		6:
			// Entry action
			IF (stStatemachine.uinState_old <> stStatemachine.uinState) THEN
				//*********************************************************
				// file close
				fbFileClose.sNetId := ''; // only local access
				fbFileClose.hFile := fbFileOpen.hFile; // only local access
				fbFileClose.tTimeout := T#3S;
				fbFileClose(bExecute:= FALSE);
				fbFileClose(bExecute:= TRUE);
				udiWaitFileCloseCycles := 0;
					
				 stStatemachine.uinState_old := stStatemachine.uinState;
			END_IF
				
			// wait UNTIL closed
			IF (fbFileClose.bBusy) THEN
				udiWaitFileCloseCycles := udiWaitFileCloseCycles + 1;
				fbFileClose(bExecute:=FALSE);
			ELSE
				IF fbFileClose.bError THEN
					strInfo := 'template/config file close failed';
					Out_udiStatus := fbFileClose.nErrId;
					RETURN;
				END_IF
				
				// delocate memory
				__DELETE(pDelReadPointer);
				
				// allocat for temporary item list
				// nbr of items * size for value output + nbf of items * Pre- and Post - Text
				// with this calculation is the buffer normally greater than necessary
				// cMAX_ITEM_CHAR has to be defined for worst case (big 4-byt values, date strings) so big
				udiTmpLen := (In_pstSysInfo^.stItemInfo.uinActNbrOfItems*FileLc.cMAX_ITEM_CHAR) + (In_pstSysInfo^.stItemInfo.uinActNbrOfItems*FileLc.cPRE_POST_TEXTLEN);
				In_pstSysInfo^.p_bytTmpRecordText := M_AllocMEM(In_SizeOfBuffer:=UDINT_TO_UINT(udiTmpLen));
				IF (In_pstSysInfo^.p_bytTmpRecordText=TC3_MEMMAN.NULL) THEN
					strInfo := 'template/config file: alloc memory for temp record text failed';
					Out_udiStatus := FileLc.cERR_ALLOC_MEMORY;
					RETURN;
				END_IF
				In_pstSysInfo^.udiTmpRecordSize := udiTmpLen;
				
				// allocat for temporary file buffer
				udiTmpLen := udiTmpLen*FileLc.cMAX_RECORDS_IN_FILE_BUF;
				In_pstSysInfo^.stFileHandler.p_bytTmpFileBuffer := M_AllocMEM(In_SizeOfBuffer:=UDINT_TO_UINT(udiTmpLen));
				IF (In_pstSysInfo^.stFileHandler.p_bytTmpFileBuffer=TC3_MEMMAN.NULL) THEN
					strInfo := 'template/config file: alloc memory for temp file buffer failed';
					Out_udiStatus := FileLc.cERR_ALLOC_MEMORY;
					RETURN;
				END_IF
				In_pstSysInfo^.stFileHandler.udiTmpFileBufferSize := udiTmpLen;
				stStatemachine.uinState := stStatemachine.uinState  + 1;
			END_IF
			
		
		7:
			stStatemachine.usiInitDone := 1;
			Out_bolDone := TRUE;
			strInfo := 'template/config file: successfully parsed';
			Out_udiStatus := 0;
	END_CASE
END_IF
bolExecute_old := In_bolExecute;

METHOD FB_exit : BOOL
VAR_INPUT
	bInCopyCode : BOOL; // if TRUE, the exit method is called for exiting an instance that is copied afterwards (online change).
END_VAR
__DELETE(pDelReadPointer);
END_METHOD

METHOD PROTECTED M_AllocMEM : POINTER TO BYTE

VAR_INPUT
	In_SizeOfBuffer : UINT; // Byte size of quee to allocate
END_VAR
// Debug counter
M_AllocMEM := __NEW(BYTE,In_SizeOfBuffer);

// check if allocate memory is ok
IF (M_AllocMEM=TC3_MEMMAN.NULL) THEN
	M_AllocMEM := TC3_MEMMAN.NULL;
ELSE
	Tc2_System.MEMSET(M_AllocMEM,0,In_SizeOfBuffer); // init with zero.
END_IF
END_METHOD

METHOD M_ReleaseAllMEM : BOOL
VAR_INPUT
	In_pstSysInfo : POINTER TO T_FileLc_SysInfo;
END_VAR
VAR
	pDelPointer : POINTER TO BYTE;
END_VAR
// no usage at the moment -> with handle shutdown sequence no easy to remove every thing in the right order


// the other allocated memory has to be deallocated by FB_FileLC! on exit this methode should be called from FB_FileLC!
IF (In_pstSysInfo<>TC3_MEMMAN.NULL) THEN
	__DELETE(In_pstSysInfo^.p_bytHeaderText);
	__DELETE(In_pstSysInfo^.p_bytFooterText);
	FOR ii:=0 TO Queue.cMAX_NR_OF_TASKS BY 1 DO
		IF (In_pstSysInfo^.stItemInfo.a_p_bytItemDataList[ii]<>TC3_MEMMAN.NULL) THEN
			pDelPointer := In_pstSysInfo^.stItemInfo.a_p_bytItemDataList[ii];
			__DELETE(pDelPointer);
			In_pstSysInfo^.stItemInfo.a_p_bytItemDataList[ii] := 0;
		END_IF
	END_FOR
	__DELETE(In_pstSysInfo^.stItemInfo.p_bytItemCfgList);
	__DELETE(In_pstSysInfo^.p_bytTmpRecordText);
	__DELETE(In_pstSysInfo^.stFileHandler.p_bytTmpFileBuffer);
	__DELETE(pDelReadPointer);
END_IF
END_METHOD

END_FUNCTION_BLOCK

// POUs/Utility/strstr
FUNCTION strstr : POINTER TO BYTE
VAR_INPUT
	In_pStr: POINTER TO BYTE; // string which should include search string
	In_pStrSearch: POINTER TO BYTE; // search string
	In_bolAddStrSearchLen : BOOL; // add to result search STRING length
END_VAR
VAR
	p_bytStr : POINTER TO BYTE;
	chrStr : STRING(1) := '';
	p_bytStrSearch : POINTER TO BYTE;
	chrStrSearch : STRING(1) := '';
	ii : UINT;
	jj : UINT;
	p_bytAdressStr : POINTER TO BYTE;
	p_bytAdressStrSearch : POINTER TO BYTE;
END_VAR

(*char *strstr(const char *s1, const char *s2);

Description
Locates the first occurence in the string pointed to by s1 of the sequence of characters in the string pointed to by s2 (excluding the terminating null character). 


Returns
Returns a pointer to the located string segment, or a null pointer if the string s2 is not found. If s2 points to a string with zero length, the s1 is returned. 
*)

// invalid input pointer check
IF ((In_pStr=TC3_MEMMAN.NULL) OR (In_pStrSearch=TC3_MEMMAN.NULL)) THEN
	strstr := TC3_MEMMAN.NULL; // input strings not defined
	RETURN;
END_IF


ii :=0;
p_bytAdressStr := In_pStr;
p_bytStr := p_bytAdressStr;
WHILE (p_bytStr^ <> 0) DO // zero terminated string
	p_bytAdressStr := In_pStr + ii*SIZEOF(In_pStr^); // pointer increment
	p_bytStr := p_bytAdressStr;
	chrStr :=Tc2_System.F_ToCHR(c:= p_bytStr^); // for debugging watch value
	
	jj := 0;
	p_bytAdressStrSearch := In_pStrSearch;
	p_bytStrSearch := p_bytAdressStrSearch;

	WHILE (p_bytStr^ = p_bytStrSearch^) DO
		
		// char/byte matches compare next
		p_bytAdressStrSearch := In_pStrSearch + jj*SIZEOF(In_pStrSearch^); // pointer increment
		p_bytStrSearch := p_bytAdressStrSearch;
		chrStrSearch := Tc2_System.F_ToCHR(c:= p_bytStrSearch^); // for debugging watch value
		
		// end of string found->search string matches
		IF (p_bytStrSearch^=0) THEN// zero terminated string
			IF (In_bolAddStrSearchLen=TRUE) THEN// add to result search STRING length
				strstr := p_bytAdressStr + jj*SIZEOF(In_pStr^); // return start adress of next byte after search string
			ELSE
				strstr := p_bytAdressStr; // return start adress of match search string
			END_IF
			
			RETURN;
		END_IF
		
		p_bytStr := p_bytAdressStr + jj*SIZEOF(In_pStr^);
		chrStr :=Tc2_System.F_ToCHR(c:= p_bytStr^); // for debugging watch value
		jj := jj + 1;
	END_WHILE
	ii := ii + 1;
END_WHILE

strstr := Tc3_MemMan.NULL; // return null adress search string not found in string

END_FUNCTION

// POUs/Utility/Logger/FileLc/FB_FileLcTest
FUNCTION_BLOCK FB_FileLcTest
VAR_INPUT
	In_p_fbBasLog: POINTER TO FB_BasLog; // only one central FB_BasLog instance allowed per PLC!!!
	In_p_fbFileLC: POINTER TO FB_FileLc; // only one central FB_FileLc instance allowed per PLC!!!
	In_strPath: STRING(FileLc.cPATH_LENGTH); //'C:\Vistaprint\Log\'
	In_strCfgFileName: STRING(FileLc.cFILENAME_LENGTH); // 'StateLogTest.cfg'
END_VAR
VAR_OUTPUT
	Out_bolInitDone : BOOL;
	Out_udiStatus : UDINT;
END_VAR
VAR
	bolGetFirstHandle : BOOL;
	bolDone : BOOL;
	udiInitStatus : UDINT;
	udiStatus : UDINT;
	pHandle : POINTER TO T_FileLc_SysInfo;
	// for test send
	pHandleBaseLog : POINTER TO T_Bl_LibHandleRow;
	uinGetHandleBaseLogStatus : UINT;
	intDoWrite : INT;
	dinPar1 : DINT;
	strText1 : STRING(30):='Controller 1';
	strText2 : STRING(30):='Alarm sub info';
	uinWriteStatus : UINT;
	bolStressTest : BOOL;
	fbRAND : DRAND;
	uinActFLcClientIdx : UINT; // file client index for init
END_VAR

(*__________________________________________________________________________________________________
¦	
¦	Vistaprint Schweiz GmbH
¦	CH - 8401 Winterthur
¦
¦	www.vistaprint.ch - info@vistaprint.ch
¦___________________________________________________________________________________________________

Function desription:
Function block capsule the logger file client call for tests.

History:
Version		Date			Author		Comment
---------------------------------------------------------------------------------------------------
0.00.1		27.10.2014		AVME/KVO	Start history
___________________________________________________________________________________________________*)

IF (In_p_fbFileLC<>TC3_MEMMAN.NULL) THEN // check if pointer valid
	
	// system init onetime after start up
	IF (Out_bolInitDone=FALSE) THEN
		In_p_fbFileLC^.M_Init(In_bolExecute := TRUE,In_p_uinFLcIdx := ADR(uinActFLcClientIdx),In_strCfgFileName:=In_strCfgFileName ,In_strPath:= In_strPath,In_p_fbBasLog := In_p_fbBasLog,Out_pHandle=>pHandle,Out_udiStatus=>udiInitStatus,Out_bolDone=>bolDone);
		IF (bolDone OR (udiInitStatus<>0)) THEN
			// negative edge -> reinit possibel and release init next file client!!!
			In_p_fbFileLC^.M_Init(In_bolExecute := FALSE,In_p_uinFLcIdx := ADR(uinActFLcClientIdx),In_strCfgFileName:=In_strCfgFileName,In_strPath:=In_strPath,In_p_fbBasLog := In_p_fbBasLog);
			Out_bolInitDone := TRUE;
		END_IF
	ELSE
		IF ((pHandle<>TC3_MEMMAN.NULL) AND (udiInitStatus=0)) THEN	// valid pointer => init ok
			// cyclic call of file client - alarm generation in application if status not ok???
			udiStatus := In_p_fbFileLC^.M_Cyclic(In_pHandle:=pHandle);
			
			// *******************************************************************************************************************************************
			// only for sending test logs!!!
			// get write handle for tests
			IF (bolGetFirstHandle=FALSE) THEN
				uinGetHandleBaseLogStatus := In_p_fbBasLog^.M_GetHandle(Out_pHandle=>pHandleBaseLog);// fbBasLog global defined base log system fub (only once per system)
				bolGetFirstHandle := TRUE;
			END_IF
			
			// write test state log entries
			IF (pHandleBaseLog<>TC3_MEMMAN.NULL) AND (intDoWrite>0) THEN
				intDoWrite := intDoWrite - 1;
				dinPar1 := dinPar1 + 1;
				uinWriteStatus := In_p_fbBasLog^.M_Log(In_pHandle:=pHandleBaseLog,In_udiLogType:=BasLog.cLOGTYPE_STATELOG,In_intCtrlID:=11,In_strText1:=strText1,In_strText2:=strText2,In_dinPar1:=dinPar1,In_dinPar2:=0,In_dinPar3:=0,In_dinPar4:=0) ;
			END_IF
			IF (bolStressTest) THEN
				IF (intDoWrite = 0) THEN
					fbRAND();
					intDoWrite := LREAL_TO_INT(fbRAND.Num*100.0);
					uinWriteStatus := In_p_fbBasLog^.M_Log(In_pHandle:=pHandleBaseLog,In_udiLogType:=BasLog.cLOGTYPE_STATELOG,In_intCtrlID:=intDoWrite,In_strText1:=strText1,In_strText2:=strText2,In_dinPar1:=dinPar1,In_dinPar2:=0,In_dinPar3:=0,In_dinPar4:=0) ;
				END_IF
			END_IF
			// *******************************************************************************************************************************************
		END_IF;		
	END_IF

	// out for failures
	IF (udiInitStatus<>0)THEN
		Out_udiStatus := udiInitStatus;
	ELSE
		Out_udiStatus := udiStatus;
	END_IF
END_IF

END_FUNCTION_BLOCK

// POUs/Utility/Queue/FB_QueueTest_Receiver
FUNCTION_BLOCK FB_QueueTest_Receiver
VAR_INPUT
	In_p_fbQueue: POINTER TO FB_Queue; // only one central FB_QUEUE instance allowed per PLC!!!
END_VAR
VAR_OUTPUT
END_VAR
VAR
	stData : T_Queue_TestData;
	bolInit : BOOL := FALSE;
	pQueueHandle : POINTER TO T_Queue_SysInfo;
	pQueueHandleRead : POINTER TO T_Queue_Info;
	uinInitStatus : UINT;
	uinGetHandleStatus :UINT;
	uinReadStatus : UINT;
	ii:UINT;
	udiRxCounter : UDINT;
END_VAR

(*__________________________________________________________________________________________________
¦	
¦	Vistaprint Schweiz GmbH
¦	CH - 8401 Winterthur
¦
¦	www.vistaprint.ch - info@vistaprint.ch
¦___________________________________________________________________________________________________

Function desription:
Example and test programm for testing the queue system - read data from queue

History:
Version		Date			Author		Comment
---------------------------------------------------------------------------------------------------
0.00.1		14.07.2014		AVME/KVO	Start history
___________________________________________________________________________________________________*)

// system init onetime after start up
IF (bolInit=FALSE) THEN
	//init queue system, one time should be called per queue system
	In_p_fbQueue^.M_Init(In_strQueueName:='bReceiver',In_uinNrOfElement := 25, In_udiSizeOfElement:= SIZEOF(stData),In_uinMode:=0,Out_pHandle=>pQueueHandle,Out_uinStatus=>uinInitStatus);
	
	// for every task class has to call this methode handle is needed for read
	uinGetHandleStatus := In_p_fbQueue^.M_GetHandle(In_strQueueName:='bReceiver',Out_pQueueHandle=>pQueueHandleRead);
	bolInit := TRUE;
END_IF

// because more than one task function writes to the logsystem it is better to read out more than one elment per cycle!
FOR ii:=0 TO 9 BY 1 DO
	uinReadStatus := In_p_fbQueue^.M_Read(In_pQueueHandle:=pQueueHandleRead,In_pData:=ADR(stData));
	IF (uinReadStatus<>0) THEN
		EXIT;
	END_IF
	udiRxCounter := udiRxCounter + 1;
END_FOR

END_FUNCTION_BLOCK

// POUs/Utility/Queue/FB_QueueTest_Sender
FUNCTION_BLOCK FB_QueueTest_Sender
VAR_INPUT
	In_p_fbQueue: POINTER TO FB_Queue; // only one central FB_QUEUE instance allowed per PLC!!!
END_VAR
VAR_OUTPUT
END_VAR
VAR
	stData : T_Queue_TestData;
	bolInit : BOOL := FALSE;
	pQueueHandle : POINTER TO T_Queue_Info;
	uinGetHandleStatus : UINT;
	uinWriteStatus :UINT;
	uinDoWrite : UINT;
END_VAR

(*__________________________________________________________________________________________________
¦	
¦	Vistaprint Schweiz GmbH
¦	CH - 8401 Winterthur
¦
¦	www.vistaprint.ch - info@vistaprint.ch
¦___________________________________________________________________________________________________

Function desription:
Example and test programm for testing the queue system - write data in queue

History:
Version		Date			Author		Comment
---------------------------------------------------------------------------------------------------
0.00.1		14.07.2014		AVME/KVO	Start history
___________________________________________________________________________________________________*)

// system init onetime after start up
IF (bolInit=FALSE) THEN
	uinGetHandleStatus := In_p_fbQueue^.M_GetHandle(In_strQueueName:='bReceiver',Out_pQueueHandle=>pQueueHandle);
	
	// init write struct
	stData.strName := 'Daten';
	stData.udiAdress := 1;
	stData.udiDataLen := 2;
	stData.usiDataTyp:= 3;
	stData.udiDimension := 4;
	bolInit := TRUE;
END_IF

// number of cycles to write
IF (uinDoWrite>0) THEN
	uinDoWrite := uinDoWrite - 1;
	uinWriteStatus := In_p_fbQueue^.M_Write(In_pQueueHandle:= pQueueHandle,In_pData:= ADR(stData));
	stData.udiAdress := stData.udiAdress + 1;
END_IF

END_FUNCTION_BLOCK

// POUs/Utility/SaberLogger/helper/cycle_Logger
FUNCTION cycle_Logger : BOOL
VAR_INPUT
	pLogger			: POINTER TO T_LoggerSendData;
END_VAR
VAR
END_VAR

pLogger^.fbFifo();

END_FUNCTION

// POUs/Utility/SaberLogger/helper/init_Logger
FUNCTION init_Logger : BOOL
VAR_INPUT
	pLogger			: POINTER TO T_LoggerSendData;
END_VAR
VAR
END_VAR

pLogger^.fbDataChannel.InitChannel(SIZEOF(pLogger^.rDataChannelItem), ADR(pLogger^.rDataChannelItem));
pLogger^.fbFifo.DataChannel := ADR(pLogger^.fbDataChannel);
pLogger^.fbFifo.FreeDataPointer := TRUE;
pLogger^.fbFifo.Enable := TRUE;

END_FUNCTION

// POUs/Utility/SaberLogger/FB_LoggerSendDch
FUNCTION_BLOCK FB_LoggerSendDch EXTENDS FB_DataChannelSendBase IMPLEMENTS I_DataChannelSend
VAR
	/// Saber Inteface Variables
	/// -----------------------------------------------------------------
	m_pOutputData: POINTER TO T_Logger_DCH;
END_VAR

SUPER^();

{attribute 'object_name' := 'InitChannel'}
METHOD InitChannel : BOOL
VAR_INPUT
	udiDataSize: UDINT;
	pOutputData: POINTER TO BYTE;
END_VAR
InitChannel := FALSE;

IF udiDataSize > 0 THEN
	IF pOutputData <> TC3_MEMMAN.NULL THEN
		m_uinDataSize := udiDataSize;
		m_pOutputData := pOutputData;
		m_eState := E_PlcSaberDHCState.Init;
		InitChannel := TRUE;
	END_IF
END_IF
END_METHOD

{attribute 'object_name' := 'SendData'}
METHOD SendData : BOOL
VAR_INPUT
	udiDataSize: UDINT;
	pData: POINTER TO BYTE;
END_VAR
SendData := FALSE;

IF m_eState = E_PlcSaberDHCState.WaitForJob THEN
	IF (udiDataSize > 0 ) AND (pData <> TC3_MEMMAN.NULL) THEN
		TC2_SYSTEM.MEMCPY(destAddr := m_pOutputData, srcAddr := pData, n := udiDataSize);
		m_eState := E_PlcSaberDHCState.SendData;	
		SendData := TRUE;
	END_IF	
END_IF
END_METHOD

END_FUNCTION_BLOCK

// POUs/Utility/callAllCtrlInit
FUNCTION callAllCtrlInit : BOOL
VAR_INPUT
	pCtrlInst			: POINTER TO POINTER TO FB_CtrlBase;
	uinCtrlInstLength	: UINT;
END_VAR
VAR
	uinIdx	: UINT;
END_VAR

FOR uinIdx := 0 TO uinCtrlInstLength DO
	IF pCtrlInst[uinIdx] <> 0 THEN
		pCtrlInst[uinIdx]^.CtrlInit(); // init ctrl and add childs
	END_IF
END_FOR

END_FUNCTION

// POUs/Utility/getInBol
FUNCTION getInBol : BOOL
VAR_INPUT
	bol_GlobalEnableForce: BOOL;
	p_Input: POINTER TO T_Ctrl_IoBool;
END_VAR

p_Input^.state := p_Input^.map;

IF (p_Input^.EnForce AND bol_GlobalEnableForce) THEN
	p_Input^.intern := p_Input^.force;
ELSE
	p_Input^.intern := p_Input^.map;
END_IF;

getInBol := p_Input^.intern;

END_FUNCTION

// POUs/Utility/getInBolDebounced
FUNCTION getInBolDebounced : BOOL
VAR_INPUT
	bol_GlobalEnableForce: BOOL;
	udiSample_ms: UDINT;		// Sample time from me.FUBInfo.udiSample_ms
	udiDebounceTime_ms: UDINT;	// Wait time for debouncing in ms
	p_Input: POINTER TO T_Ctrl_IoBoolDebounced;
END_VAR

// The input is accepted only after the debounce time (udiDebounceTime_ms)
// If the signal changes during this time, the timer will be restarted

IF (p_Input^.EnForce AND bol_GlobalEnableForce) THEN	// Forced signal, no debouncing neccessary
	p_Input^.intern := p_Input^.force;
ELSE													// Debounce signal
	IF p_Input^.state <> p_Input^.map THEN
		p_Input^.udinDebouncedTimeCounter_ms := 0;
	END_IF
	IF p_Input^.udinDebouncedTimeCounter_ms < udiDebounceTime_ms THEN
		p_Input^.udinDebouncedTimeCounter_ms := p_Input^.udinDebouncedTimeCounter_ms + udiSample_ms;
	ELSE
		p_Input^.intern := p_Input^.map;		
	END_IF
END_IF;

p_Input^.state := p_Input^.map;

getInBolDebounced := p_Input^.intern;

END_FUNCTION

// POUs/Utility/getInInt
FUNCTION getInInt : INT
VAR_INPUT
	bol_GlobalEnableForce: BOOL;
	p_Input: POINTER TO T_Ctrl_IoInt;
END_VAR

p_Input^.state := p_Input^.map;

IF (p_Input^.EnForce AND bol_GlobalEnableForce) THEN
	p_Input^.intern := p_Input^.force;
ELSE
	p_Input^.intern := p_Input^.map;
END_IF;

getInInt := p_Input^.intern;

END_FUNCTION

// POUs/Utility/getInUint
FUNCTION getInUint : UINT
VAR_INPUT
	bol_GlobalEnableForce		: BOOL;
	p_Input						: POINTER TO T_Ctrl_IoUint;
END_VAR
VAR
END_VAR

p_Input^.state := p_Input^.map;

IF (p_Input^.EnForce AND bol_GlobalEnableForce) THEN
	p_Input^.intern := p_Input^.force;
ELSE
	p_Input^.intern := p_Input^.map;
END_IF;

getInUint := p_Input^.intern;

END_FUNCTION

// POUs/Utility/getInUsint
FUNCTION getInUsint : USINT
VAR_INPUT
	bol_GlobalEnableForce		: BOOL;
	p_Input						: POINTER TO T_Ctrl_IoUsint;
END_VAR
VAR
END_VAR

p_Input^.state := p_Input^.map;

IF (p_Input^.EnForce AND bol_GlobalEnableForce) THEN
	p_Input^.intern := p_Input^.force;
ELSE
	p_Input^.intern := p_Input^.map;
END_IF;

getInUsint := p_Input^.intern;

END_FUNCTION

// POUs/Utility/initAllCtrl
FUNCTION initAllCtrl : BOOL
VAR_INPUT
	pCtrlInst			: POINTER TO POINTER TO FB_CtrlBase;
	pBasLogFB			: POINTER TO FB_BasLog;
	pAlarmCtrl			: POINTER TO FB_Alm_Man;
	uinCtrlInstLength	: UINT;
END_VAR
VAR
	uinIdx	: UINT;
END_VAR

FOR uinIdx := 0 TO uinCtrlInstLength DO
	IF pCtrlInst[uinIdx] <> 0 THEN
		IF (pAlarmCtrl<>0) THEN
			pCtrlInst[uinIdx]^.AlarmCtrl := pAlarmCtrl; // add alarm manager interface/pointer
		END_IF
		IF (pBasLogFB<>0) THEN
			pCtrlInst[uinIdx]^.BaseLog := pBasLogFB; // add base logger interface/pointer
		END_IF
		pCtrlInst[uinIdx]^.CtrlInit(); // init ctrl and add childs
	END_IF
END_FOR

END_FUNCTION

// POUs/Utility/ScaleINT
FUNCTION ScaleINT : INT //Output signal.
VAR_INPUT
	x: INT; 	// Input signal. Allowed values: -32768..+32767.
	x1 : INT;	// Abscissa for the 1st coordinate. Allowed values: -32768..+32767
	x2 : INT;	// Abscissa for the 2nd coordinate. Allowed values: -32768..+32767.
	y1 : INT;	// Ordinate for the 1st coordinate. First limit of the value range. Allowed values: –32768..+32767.
	y2: INT;	// Ordinate for the 2nd coordinate. Second limit of the value range. Allowed values: -32768..+32767.
END_VAR
VAR
END_VAR


(*	IF x1 = x2, THEN 0 is output *)

// Scale value 
IF (x1=x2) THEN // -> zero division!
	ScaleINT := 0;
ELSE
	ScaleINT := (((x - x1) * (y2-y1))/(x2-x1)) + y1;
END_IF

END_FUNCTION

// POUs/Utility/setAllCtrlAlarmFB
FUNCTION setAllCtrlAlarmFB : BOOL
VAR_INPUT
	pCtrlInst			: POINTER TO POINTER TO FB_CtrlBase;
	pAlarmCtrl			: POINTER TO FB_Alm_Man;
	uinCtrlInstLength	: UINT;
END_VAR
VAR
	uinIdx	: UINT;
END_VAR

FOR uinIdx := 0 TO uinCtrlInstLength DO
	IF pCtrlInst[uinIdx] <> 0 THEN
		pCtrlInst[uinIdx]^.AlarmCtrl := pAlarmCtrl;
	END_IF
END_FOR

END_FUNCTION

// POUs/Utility/setAllCtrlBasLogFB
FUNCTION setAllCtrlBasLogFB : BOOL
VAR_INPUT
	pCtrlInst			: POINTER TO POINTER TO FB_CtrlBase;
	pBasLogFB			: POINTER TO FB_BasLog;
	uinCtrlInstLength	: UINT;
END_VAR
VAR
	uinIdx	: UINT;
END_VAR

FOR uinIdx := 0 TO uinCtrlInstLength DO
	IF pCtrlInst[uinIdx] <> 0 THEN
		pCtrlInst[uinIdx]^.BaseLog := pBasLogFB;
	END_IF
END_FOR

END_FUNCTION

// POUs/Utility/setOutBol
FUNCTION setOutBol : BOOL
VAR_INPUT
	bol_GlobalEnableForce: BOOL;
	p_Output: POINTER TO T_Ctrl_IoBool;
END_VAR

// Copy real values
p_Output^.state := p_Output^.intern;

IF (p_Output^.EnForce AND bol_GlobalEnableForce) THEN
	p_Output^.map := p_Output^.force;
ELSE
	p_Output^.map := p_Output^.intern;
END_IF;

setOutBol := p_Output^.map;

END_FUNCTION

// POUs/Utility/setOutInt
FUNCTION setOutInt : INT
VAR_INPUT
	bol_GlobalEnableForce: BOOL;
	p_Output: POINTER TO T_Ctrl_IoInt;
END_VAR

// Copy real values
p_Output^.state := p_Output^.intern;

IF (p_Output^.EnForce AND bol_GlobalEnableForce) THEN
	p_Output^.map := p_Output^.force;
ELSE
	p_Output^.map := p_Output^.intern;
END_IF;

setOutInt := p_Output^.map;

END_FUNCTION

// POUs/Utility/setOutUint
FUNCTION setOutUint : UINT
VAR_INPUT
	bol_GlobalEnableForce	: BOOL;
	p_Output				: POINTER TO T_Ctrl_IoUint;
END_VAR
VAR
END_VAR

// Copy real values
p_Output^.state := p_Output^.intern;

IF (p_Output^.EnForce AND bol_GlobalEnableForce) THEN
	p_Output^.map := p_Output^.force;
ELSE
	p_Output^.map := p_Output^.intern;
END_IF;

setOutUint := p_Output^.map;

END_FUNCTION

// POUs/Utility/setOutUsint
FUNCTION setOutUsint : USINT
VAR_INPUT
	bol_GlobalEnableForce	: BOOL;
	p_Output				: POINTER TO T_Ctrl_IoUsint;
END_VAR
VAR
END_VAR

// Copy real values
p_Output^.state := p_Output^.intern;

IF (p_Output^.EnForce AND bol_GlobalEnableForce) THEN
	p_Output^.map := p_Output^.force;
ELSE
	p_Output^.map := p_Output^.intern;
END_IF;

setOutUsint := p_Output^.map;

END_FUNCTION
